// Mitsubishi GX Works2 project: hmi_led_fx2n   PLC: FX2N/FX2NC

PROGRAM MAIN
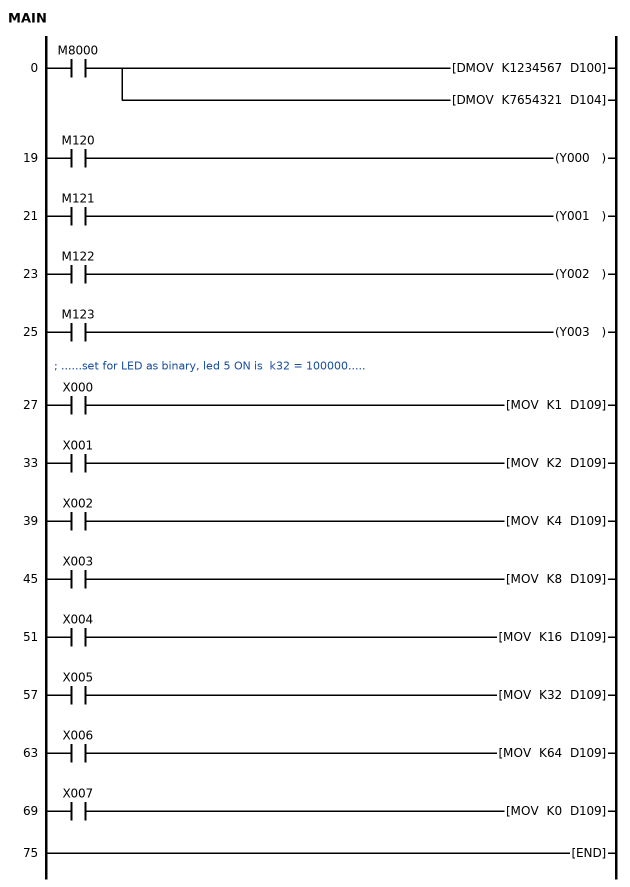
0     LD      M8000
      DMOV    K1234567 D100
      DMOV    K7654321 D104
19    LD      M120
      OUT     Y000
21    LD      M121
      OUT     Y001
23    LD      M122
      OUT     Y002
25    LD      M123
      OUT     Y003
; ......set for LED as binary, led 5 ON is  k32 = 100000.....
27    LD      X000
      MOV     K1 D109
33    LD      X001
      MOV     K2 D109
39    LD      X002
      MOV     K4 D109
45    LD      X003
      MOV     K8 D109
51    LD      X004
      MOV     K16 D109
57    LD      X005
      MOV     K32 D109
63    LD      X006
      MOV     K64 D109
69    LD      X007
      MOV     K0 D109
75    END
END_PROGRAM
